// TIA Portal V17 export
// export: Created 2025-03-05T08:01:53.3705552Z, ExportSetting WithDefaults, DisplayName Totally Integrated Automation Portal, DisplayVersion V17 Update 8, DisplayName TIA Portal Openness, DisplayVersion V17 Update 8, DisplayName TIA Portal Version Control Interface, DisplayVersion V17, DisplayName SINAMICS Startdrive Advanced, DisplayVersion V17 SP2, DisplayName SINAMICS Startdrive G110M, G120, G120C, G120D, G120P, G115D, DisplayVersion V17 SP2, DisplayName SINAMICS Startdrive G130, G150, S120, S150, SINAMICS MV, S210, DisplayVersion V17 SP2, DisplayName STEP 7 Professional, DisplayVersion V17 Update 8, DisplayName SINUMERIK ONE STEP 7 Toolbox, DisplayVersion V17 Update 12, DisplayName SINUMERIK 840D sl STEP 7 Toolbox, DisplayVersion V17 Update 12, DisplayName STEP 7 Safety, DisplayVersion V17 Update 6, DisplayName WinCC Advanced, DisplayVersion V17 Update 8
VAR_GLOBAL   // PLC tag table "TAGS_IO_SERVICES_CLADDING"
   "/////_PNEUMATIC_/////" AT %M8020.0 : Bool;   // /////_PNEUMATIC_/////
   PNM_S_P_CON_SENSOR_1_I AT %M8020.1 : Bool;   // PNEUMATIC SYSTEM PNEUMATIC CONNECTION 1 SENSOR INPUT NO
   PNM_S_P_CON_SENSOR_2_I AT %M8020.2 : Bool;   // PNEUMATIC SYSTEM PNEUMATIC CONNECTION 2 SENSOR INPUT NO
   PNM_S_PRESS_PRSNT_I AT %I51.1 : Bool;   // PNEUMATIC SYSTEM PRESSURE PRESENT INPUT NO
   PNM_S_PRSSRZD_I AT %I51.2 : Bool;   // PNEUMATIC SYSTEM PRESSURIZED INPUT NO
   PNM_S_DRV_UBLCKD_I AT %M8020.5 : Bool;   // PNEUMATIC SYSTEM DRIVE UNBLOCKED INPUT NC
   PNM_S_PR_MQL_AIR_I AT %M8020.6 : Bool;   // PNEUMATIC SYSTEM MQL COMPRESSED AIR INPUT NO
   PNM_S_PR_U01_GRIPPER_I AT %I62.0 : Bool;   // PNEUMATIC SYSTEM UNIT 01 GRIPPER PRESSURIZED INPUT NO
   PNM_S_PR_U01_LABERINT_I AT %I62.1 : Bool;   // PNEUMATIC SYSTEM IUNIT 01 LABERINT PRESSURIZED INPUT NO
   PNM_S_PR_U01_UP_TABLE_I AT %I62.2 : Bool;   // PNEUMATIC SYSTEM UNIT 01 UPPER TABLE PRESSURIZED INPUT NO
   PNM_S_PR_U01_DOWN_TABLE_I AT %I62.3 : Bool;   // PNEUMATIC SYSTEM UNIT 01 LOWER TABLE PRESSURIZED INPUT NO
   PNM_S_PR_U01_X_CART_I AT %I62.4 : Bool;   // PNEUMATIC SYSTEM UNIT 01 AXIS X13 CART PRESSURIZED INPUT NO
   PNM_S_PR_U02_GRIPPER_I AT %I1062.0 : Bool;   // PNEUMATIC SYSTEM UNIT 02 GRIPPER PRESSURIZED INPUT NO
   PNM_S_PR_U02_LABERINT_I AT %I1062.1 : Bool;   // PNEUMATIC SYSTEM IUNIT 02 LABERINT PRESSURIZED INPUT NO
   PNM_S_PR_U02_UP_TABLE_I AT %I1062.2 : Bool;   // PNEUMATIC SYSTEM UNIT 02 UPPER TABLE PRESSURIZED INPUT NO
   PNM_S_PR_U02_DOWN_TABLE_I AT %I1062.3 : Bool;   // PNEUMATIC SYSTEM UNIT 02 LOWER TABLE PRESSURIZED INPUT NO
   PNM_S_PR_U02_X_CART_I AT %I1062.4 : Bool;   // PNEUMATIC SYSTEM UNIT 02 AXIS X13 CART PRESSURIZED INPUT NO
   PNM_S_PR_U02_ST3_MEAS AT %I1062.5 : Bool;   // PNEUMATIC SYSTEM UNIT 02 STATION 3 MEASUREMENT PRESSURIZED INPUT NO
   PNM_S_FLOW_SENSOR_I AT %MW8024 : Word;   // PNEUMATIC SYSTEM FLOW SENSOR INPUT
   PNM_S_TEMP_SENSOR_I AT %MW8026 : Word;   // PNEUMATIC SYSTEM TEMPERATURE SENSOR INPUT
   PNM_M_VLV_ON_Q AT %Q50.0 : Bool;   // SWITCH-ON PNEUMATIC SYSTEM
   PNM_M_VLV_ON2_Q AT %M8027.0 : Bool;   // SWITCH-ON PNEUMATIC SYSTEM 2
   PNM_S_P_CON_SENSOR_1_Q AT %M8027.1 : Bool;   // PNEUMATIC SYSTEM PNEUMATIC CONNECTION 1 SENSOR OUTPUT
   PNM_S_P_CON_SENSOR_2_Q AT %M8027.2 : Bool;   // PNEUMATIC SYSTEM PNEUMATIC CONNECTION 2 SENSOR OUTPUT
   PNM_PRSZTN_ON_Q AT %Q51.0 : Bool;   // SWITCH-ON PNEUMATIC PRESSURIZATION
   PNM_PRSZTN_OFF_Q AT %M8027.3 : Bool;   // SWITCH-OFF PNEUMATIC PRESSURIZATION
   PNM_DRIVE_UNBLCK_Q AT %M8027.4 : Bool;   // UNBLOCK PNEUMATIC DRIVE
   "/////_LUBRICATION_/////" AT %M8040.0 : Bool;   // /////_LUBRICATION_/////
   LB_PMP_BREAKER_I AT %M8040.1 : Bool;   // LUBRICATION PUMP CIRCUIT BREAKER INPUT NC
   LB_U_LOW_LEVEL_ALM_I AT %M8040.2 : Bool;   // LUBRICATION UNIT LOW LEVEL ALARM INPUT NC
   LB_U_FILTER_CLOGGED_ALM_I AT %M8040.3 : Bool;   // LUBRICATION UNIT FILTER CLOGGED ALARM INPUT NC
   LB_U_FIXTURE_PRESS_RCHD_I AT %M8040.4 : Bool;   // LUBRICATION UNIT CLAMPING FIXTURE LUBRICATION PRESSURE REACHED INPUT NO
   LB_U01_PRESS_RCHD_I AT %M8040.5 : Bool;   // LUBRICATION UNIT UNIT 01R LUBRICATION PRESSURE REACHED INPUT NO
   LB_U02_PRESS_RCHD_I AT %M8040.6 : Bool;   // LUBRICATION UNIT UNIT 01L LUBRICATION PRESSURE REACHED INPUT NO
   LB_U_LOW_LEVEL_PREALM_I AT %M8040.7 : Bool;   // LUBRICATION UNIT LOW LEVEL PREALARM INPUT NC
   LB_U_FILTER_CLOGGED_PREALM_I AT %M8041.0 : Bool;   // LUBRICATION UNIT FILTER CLOGGED PREALARM INPUT NC
   LB_PMP_ON_Q AT %Q42.3 : Bool;   // LUBRICATION UNIT SWITCH-ON
   LB_BRANCH_1_DONE AT %I52.0 : Bool;   // LUBRICATION BRANCH 01 DONE
   LB_BRANCH_2_DONE AT %I52.1 : Bool;   // LUBRICATION BRANCH 02 DONE
   LB_BRANCH_3_DONE AT %I52.2 : Bool;   // LUBRICATION BRANCH 03 DONE
   LB_VLV_1_ON_Q AT %Q51.1 : Bool;   // LUBRICATION UNIT SWITCH-ON BRANCH E1 VALVE
   LB_VLV_2_ON_Q AT %Q51.2 : Bool;   // LUBRICATION UNIT SWITCH-ON BRANCH E2 VALVE
   LB_VLV_3_ON_Q AT %Q51.3 : Bool;   // LUBRICATION UNIT SWITCH-ON BRANCH E3 VALVE
   "/////_COOLING_CHILLER_/////" AT %M8100.0 : Bool;   // /////_COOLING_CHILLER_/////
   COOLING_UNIT_ON AT %I37.5 : Bool;   // COOLING UNIT ON
   COOLING_UNIT_02_FLOW_CONTROL_INPUTS AT %MW8102 : Word;   // COOLING SYSTEM UNIT 02 FLOW CONTROL INPUTS
   COOLING_UNIT_02_FLOW_CONTROL_OUTPUTS AT %MW8104 : Word;   // COOLING SYSTEM UNIT 02 FLOW CONTROL INPUTS
   "/////_EXTRACTION_/////" AT %M8311.0 : Bool;   // /////_EXTRACTION_/////
   U01_STA_4_EXTRAC_FLOW_PRESENT_UPPER AT %I480.2 : Bool;   // UNIT 01 STATION 4 EXTRACTION FLOW PRESENT UPPER
   U01_STA_4_EXTRAC_FLOW_PRESENT_LOWER AT %I480.3 : Bool;   // UNIT 01 STATION 4 EXTRACTION FLOW PRESENT LOWER
   U02_STA_4_EXTRAC_FLOW_PRESENT_UPPER AT %I1480.2 : Bool;   // UNIT 02 STATION 4 EXTRACTION FLOW PRESENT UPPER
   U02_STA_4_EXTRAC_FLOW_PRESENT_LOWER AT %I1480.3 : Bool;   // UNIT 02 STATION 4 EXTRACTION FLOW PRESENT LOWER
   MIST_EXTRACTION_READY AT %I45.0 : Bool;   // MIST EXTRACTION READY
   MIST_EXTRACTION_FAULT AT %I45.1 : Bool;   // MIST EXTRACTION FAULT
   MIST_EXTRACTION_REQ_FILTER_CLEAN AT %M8312.3 : Bool;   // MIST EXTRACTION REQUIRE FILTER CLEANING
   MIST_EXTRACTION_SWITCH_ON AT %Q41.0 : Bool;   // MIST EXTRACTION SWITCH ON
   MIST_EXTRACTION_MACHINE_OK AT %Q41.1 : Bool;   // MIST EXTRACTION MACHINE OK
   MIST_EXTRACTION_ALLOW_CLEANING AT %M8312.6 : Bool;   // MIST EXTRACTION ALLOW CLEANING
   "/////_PROTECTION_GAS_/////" AT %M8350.0 : Bool;
   U01_GAS_FLOW_VALUE AT %ID672 : Real;   // UNIT 01 GAS FLOW VALUE
   U01_GAS_FLOW_SET_POINT AT %QD670 : Real;   // UNIT 01 GAS FLOW SET POINT
   U01_GAS_TEMPERATURE_VALUE AT %IW676 : UInt;   // UNIT 01 GAS TEMPERATURE VALUE
   U02_GAS_FLOW_VALUE AT %ID1672 : Real;   // UNIT 02 GAS FLOW VALUE
   U02_GAS_FLOW_SET_POINT AT %QD1670 : Real;   // UNIT 02 GAS FLOW SET POINT
   U02_GAS_TEMPERATURE_VALUE AT %IW1676 : UInt;   // UNIT 02 GAS TEMPERATURE VALUE
   U02_TURN_CONTROL_1 AT %I1500.4 : Bool;   // UNIT 02 TURN CONTROL 1
   U02_TURN_CONTROL_2 AT %I1500.5 : Bool;   // UNIT 02 TURN CONTROL 2
   U02_KF1076_SAFE_VALVE_Q AT %Q1072.0 : Bool;   // UNIT 02 KF1076 SAFETY VALVE OUTPUT
   UNIT_01_PROTEC_GAS_SW_ON_Q AT %Q70.4 : Bool;   // UNIT 01 PROTECTION GAS 1 SWITCH ON OUTPUT
   AUXILIARY_COOLING_TEMP_ALARM AT %I56.0 : Bool;   // AUXILIARY COOLING TEMPERATURE ALARM
   GENERAL_GAS_PRESS_PRSNT_I AT %I51.3 : Bool;   // GENERAL GAS SYSTEM PRESSURE PRESENT INPUT
   UNIT_02_PROTEC_GAS_SW_ON_Q AT %Q1070.4 : Bool;   // UNIT 02 PROTECTION GAS 1 SWITCH ON OUTPUT
   UNIT_02_PROTEC_GAS_SW_OFF_Q AT %Q1071.4 : Bool;
   PNM_S_PR_U01_ST3_MEAS AT %M8020.7 : Bool;   // PNEUMATIC SYSTEM UNIT 01 STATION 3 MEASUREMENT PRESSURIZED INPUT NO
   COOLING_U02_LASER_INPUT_FLOW_VALUE_INPUT AT %MD8412 : DInt;   // COOLING SYSTEM UNIT 02 LASER INPUT FLOW VALUE INPUT
   COOLING_U01_LASER_INPUT_TEMP_VALUE_INPUT AT %MD8416 : DInt;   // COOLING SYSTEM UNIT 01 LASER INPUT TEMP VALUE INPUT
   COOLING_U02_LASER_INPUT_TEMP_VALUE_INPUT AT %MD8420 : DInt;   // COOLING SYSTEM UNIT 02 LASER INPUT TEMPVALUE INPUT
   COOLING_U01_LASER_INPUT_FLOW_CONTROL_ALM_I AT %I55.1 : Bool;   // COOLING SYSTEM UNIT 01 LASER INPUT FLOW CONTROL ALARM INPUT
   COOLING_U02_LASER_INPUT_TEMP_CONTROL_ALM_I AT %I55.7 : Bool;   // COOLING SYSTEM UNIT 02 LASER TEMPERATURE CONTROL ALARM INPUT
   COOLING_U01_LASER_INPUT_TEMP_CONTROL_ALM_I AT %I55.5 : Bool;   // COOLING SYSTEM UNIT 01 LASER TEMPERATURE CONTROL ALARM INPUT
   COOLING_U02_LASER_INPUT_FLOW_CONTROL_ALM_I AT %I55.3 : Bool;   // COOLING SYSTEM UNIT 02 LASER INPUT FLOW CONTROL ALARM INPUT
   COOLING_U01_LASER_TOT_OUTPUT_FLOW_VALUE_INPUT AT %ID832 : Real;   // COOLING SYSTEM UNIT 01 LASER TOTAL OUTPUT FLOW VALUE INPUT
   COOLING_U01_LASER_INPUT_FLOW_VALUE_INPUT AT %MD818 : DInt;   // COOLING SYSTEM UNIT 01 LASER INPUT FLOW VALUE INPUT
   COOLING_U01_LASER_OUTPUT_FLOW_VALUE_INPUT AT %ID836 : DInt;   // COOLING SYSTEM UNIT 01 LASER OUTPUT FLOW VALUE INPUT
   COOLING_U01_LASER_OUTPUT_TEMP_VALUE_INPUT AT %ID842 : DInt;   // COOLING SYSTEM UNIT 01 LASER OUTPUT TEMP VALUE INPUT
   COOLING_U02_LASER_TOT_OUTPUT_FLOW_VALUE_INPUT AT %ID848 : Real;   // COOLING SYSTEM UNIT 02 LASER TOTAL OUTPUT FLOW VALUE INPUT
   COOLING_U02_LASER_OUTPUT_FLOW_VALUE_INPUT AT %ID852 : DInt;   // COOLING SYSTEM UNIT 02 LASER OUTPUT FLOW VALUE INPUT
   COOLING_U02_LASER_OUTPUT_TEMP_VALUE_INPUT AT %ID858 : DInt;   // COOLING SYSTEM UNIT 02 LASER OUTPUT TEMP VALUE INPUT
   AUXILIARY_COOLING_LOW_LVL_ALARM AT %I56.4 : Bool;   // AUXILIARY COOLING LOW LEVEL ALARM
   COOLING_SECONDARY_SHIELD_SWITCH_ON AT %Q42.1 : Bool;   // UNIT 01 COOLING UNIT SWITCH ON
   COOLING_SECONDARY_BUFFER_SWITCH_ON AT %Q42.2 : Bool;   // COOLING UNIT 02 SWITCH ON
   SECUNDARY_COOLING_BUFFER_LOW_LVL_ALARM AT %I56.5 : Bool;   // SECUNDARY COOLING LOW LEVEL ALARM
   SECUNDARY_COOLING_BUFFER_TEMP_ALARM AT %I56.1 : Bool;   // SECUNDARY COOLING TEMPERATURE ALARM
   COOLING_BUFFER_FEEDBACK_ON AT %I38.7 : Bool;   // COOLING UNIT 02 FEEDBACK ON
   COOLING_UNIT_01_02_FEEDBACK_ON AT %I38.6 : Bool;   // COOLING UNIT 01 FEEDBACK ON
   MAIN_COOLING_TEMP_CONTROL_INPUTS AT %IW802 : Int;   // COOLING SYSTEM MAIN TEMPERATURE CONTROL INPUTS
   MAIN_COOLING_FLOW_CONTROL_INPUTS AT %IW800 : Int;   // COOLING SYSTEM MAIN FLOW CONTROL INPUTS
   MAIN_COOLING_TEMP_CONTROL_OUTPUTS AT %IW810 : Int;   // COOLING SYSTEM MAIN TEMPERATURECONTROL OUTPUTS
   MAIN_COOLING_FLOW_CONTROL_OUTPUTS AT %IW808 : Int;   // COOLING SYSTEM MAIN FLOW CONTROL OUTPUTS
   MAIN_COOLING_OUTPUT_FLOW_SP AT %I811.0 : Bool;   // COOLING SYSTEM MAIN OUTPUT FLOW SETPOINT
   MAIN_COOLING_INPUT_TEMP_SP AT %I803.1 : Bool;   // COOLING SYSTEM MAIN INPUT TEMP SETPOINT
   MAIN_COOLING_INPUT_FLOW_SP AT %I803.0 : Bool;   // COOLING SYSTEM MAIN INPUT FLOW SETPOINT
   MAIN_COOLING_OUTPUT_TEMP_SP AT %I811.1 : Bool;   // COOLING SYSTEM MAIN OUTPUT TEMP SETPOINT
END_VAR
